PROGRAM MAIN
VAR
END_VAR

Sum(3.4, 5.1);

END_PROGRAM

(* stored: Version 1.1.0.1, ProductVersion 3.1.4024.3
   POU MAIN: Id {09b3976b-e985-4146-9fa7-ddf97df77b95}, SpecialFunc None *)
